{attribute 'linkalways'}
{attribute 'hide_all_locals'}
FUNCTION_BLOCK ValueDtRead EXTENDS ValueBase IMPLEMENTS ValueRead
VAR
	thisValue : DT;
END_VAR

{attribute 'call_after_global_init_slot' := '1'}
{attribute 'call_after_online_change_slot' := '1'}
METHOD PROTECTED GetThisAnyType
VAR_INPUT
END_VAR
thisAnyType := ToAnyType(thisValue);
END_METHOD

METHOD GetAsType : BOOL
VAR_INPUT
	destination : __SYSTEM.AnyType;
END_VAR
GetAsType := ConvertAnyType(thisAnyType, destination);
END_METHOD

METHOD GetAsString : T_MaxString
VAR_INPUT
END_VAR
GetAsString := DT_TO_STRING(thisValue);
END_METHOD

METHOD Get : BOOL
VAR_INPUT
	destination : ANY;
END_VAR
Get := ConvertAnyType(thisAnyType, destination);
END_METHOD

METHOD FB_init : BOOL
VAR_INPUT
	bInitRetains : BOOL; // if TRUE, the retain variables are initialized (warm start / cold start)
	bInCopyCode : BOOL;  // if TRUE, the instance afterwards gets moved into the copy code (online change)
END_VAR
_ValueType := __SYSTEM.TYPE_CLASS.TYPE_DATEANDTIME;
END_METHOD

{attribute 'monitoring' := 'call'}
PROPERTY Value : DT
GET
Value := thisValue;
END_GET
END_PROPERTY

END_FUNCTION_BLOCK

(* stored: Version 1.1.0.1
   POU ValueDtRead: Id {05c5e6ba-5e26-438f-a6f6-164d04841c6b}, SpecialFunc None
   Method GetThisAnyType: Id {0807fe6e-3d1d-4c2d-a9f9-df0fcac805fe}
   Method GetAsType: Id {d2a160f9-99f9-4f9a-8631-2744de2fc6cd}
   Method GetAsString: Id {483996e3-df2e-421e-bad6-57a8b6b54552}
   Method Get: Id {37cbf016-4dd9-4ca8-a514-c6b50eb8dbf7}
   Method FB_init: Id {e94881ba-bad1-4a31-952b-53430563e6fd}
   Property Value: Id {968ac5e8-cc69-4d1f-8ba7-e6ff514ac49a}
   Get Get: Id {1682aec0-8404-401f-9ac7-16eb66e2783b} *)
